// TIA Portal V19 export
TYPE "LEXCHANGETRAY_typeSR1000ProfinetConfigeration"
// referenceDesignator: String[20]
// simActive: Bool
// simError: Int
// preRescanCounter: Int
// hwd: HW_ANY
// telegram: LEXCHANGETRAY_typeSr1000ProfinetTelegram
// stored: Access Published
   STRUCT
      referenceDesignator : String[20] := 'U3Em1IO';
      simActive : Bool;
      simError : Int;   // 仿真模拟扫码失败次数
      preRescanCounter : Int;   // 重试次数
      hwd : HW_ANY;
      telegram : "LEXCHANGETRAY_typeSr1000ProfinetTelegram";
   END_STRUCT;
END_TYPE
